// TIA Portal V20 export
// export: Created 2025-12-01T14:57:15.6741069Z, ExportSetting None, DisplayName Totally Integrated Automation Portal, DisplayVersion V20 Update 3, DisplayName TIA Portal Openness, DisplayVersion V20 Update 3, DisplayName TIA Portal Version Control Interface, DisplayVersion V20 Update 3, DisplayName STEP 7 Professional, DisplayVersion V20 Update 3, DisplayName STEP 7 Safety, DisplayVersion V20 Update 2, DisplayName WinCC Basic/Comfort/Advanced, DisplayVersion V20 Update 3, DisplayName WinCC Professional, DisplayVersion V20 Update 3, DisplayName WinCC Unified, DisplayVersion V20 Update 3
DATA_BLOCK "DB811_ColasMckeys"   // DB811
{ S7_Optimized_Access := 'FALSE' }
AUTHOR : TRACKING
NAME : 20130301
VERSION : 3.0
// stored: AutoNumber false
   VAR
      Colas_Mckey : Array[0..9999] of Struct
         UT_PrimerMckey : UInt;
      END_STRUCT;
      MckeyUT : Array[0.."CTE_MaxUTs"] of Struct
         UT_AnteriorMckey : UInt;
         UT_SiguienteMcKey : UInt;
      END_STRUCT;
   END_VAR
BEGIN
   MckeyUT[5].UT_AnteriorMckey := 1;
END_DATA_BLOCK
